(* implements non-volatile data using XML file and XML Server (max 4K) *)
FUNCTION_BLOCK FB_CX_NVData_XMLFile_4K
VAR_INPUT
	bEnable				: BOOL;		(* set TRUE to load and monitor XML data *)
	bReset				: BOOL;		(* set TRUE to reset error and re-start sequence *)
	bBackup				: BOOL;		(* set TRUE to write data to backup XML file *)
	bRestore			: BOOL;		(* set TRUE to restore data from backup XML file *)
	pSourceData			: POINTER TO BYTE;	(* pointer to source data structure *)
	nSourceBytes		: UDINT;		(* no of bytes in source data structure *)
	strXPath			: T_MaxString;	(* XPath for XML file *)
	strXMLPathFile		: T_MaxString;	(* XML file name, backup XML file will have '.bak' appended to the end *)
	tUpdateTime			: TIME;		(* update time to check for changes in memory *)
END_VAR
VAR_OUTPUT
	bNVDataInitOK		: BOOL;		(* TRUE = data loaded OK *)
	bFileWriteError		: BOOL;		(* TRUE = XML file write error *)
	bDataChanged		: BOOL;		(* TRUE = change of data detected *)
	nTotalChanges		: UDINT;	(* total number of data changes *)
END_VAR
VAR
	fbBackup			: R_TRIG;
	bBackupReq			: BOOL;
	fbRestore			: R_TRIG;
	bRestoreReq			: BOOL;

	eState				: E_CX_NVXMLState;
	fbDelayTimer		: TON;
	nRetries			: BYTE;
	fbReadXML			: FB_XmlSrvRead;
	fbMonitor			: FB_MemoryMonitor_4K;
	fbWriteXML			: FB_XmlSrvWrite;
	nOnlineChangeCount	: UDINT;
END_VAR
(*
-------------------------------------------------------------------------------------------------
Date		Version	Author	Comments
-------------------------------------------------------------------------------------------------
30/01/2015	3.00.00	PB		Initial release

-------------------------------------------------------------------------------------------------
*)

(* backup requested *)
fbBackup(CLK := bBackup);
IF fbBackup.Q = TRUE THEN

	bBackupReq := TRUE;
END_IF

(* restore requested *)
fbRestore(CLK := bRestore);
IF fbRestore.Q = TRUE THEN

	bRestoreReq := TRUE;
END_IF


CASE eState OF

	(* idle state *)
	E_CX_NVXML_IDLE:

		(* enabled*)
		IF bEnable = TRUE THEN

			(* update outputs *)
			bNVDataInitOK := FALSE;
			bFileWriteError := FALSE;

			eState := E_CX_NVXML_READXML;

		(* disabled *)
		ELSE

			(* reset outputs *)
			bNVDataInitOK := FALSE;
			bFileWriteError := FALSE;
			bDataChanged := FALSE;
			nTotalChanges := 0;

			(* reset event flags *)
			bBackupReq := FALSE;
			bRestoreReq := FALSE;
		END_IF


	(* read data *)
	E_CX_NVXML_READXML:

		(* read XML file *)
		fbReadXML(
			sNetId		:= '',
			ePath		:= PATH_GENERIC,
			nMode		:= XMLSRV_SKIPMISSING,
			pSymAddr	:= pSourceData,
			cbSymSize	:= nSourceBytes,
			sFilePath	:= strXMLPathFile,
			sXPath		:= strXPath,
			bExecute	:= TRUE,
			tTimeout	:= T#1s
		);

		(* XML read complete *)
		IF fbReadXML.bBusy = FALSE THEN

			(* XML read completed OK *)
			IF fbReadXML.bError = FALSE THEN

				(* XML file has been read at least once *)
				bNVDataInitOK := TRUE;

				eState := E_CX_NVXML_MONITOR;

			(* XML read error *)
			ELSE

				(* file access error *)
				IF fbReadXML.nErrId < 16#8000 THEN

					(* increment retry counter and wait for next read attempt *)
					nRetries := nRetries + 1;

					eState := E_CX_NVXML_RETRY;

				(* XML server error *)
				ELSE

					(* data has previously been read using XML Server *)
					IF bNVDataInitOK = TRUE THEN

						eState := E_CX_NVXML_MONITOR;

					(* data has not previously been read using XML Server *)
					ELSE

						eState := E_CX_NVXML_RESTORE;
					END_IF
				END_IF
			END_IF

			(* close off fbReadXML *)
			fbReadXML(bExecute := FALSE);
		END_IF


	(* restore backup data *)
	E_CX_NVXML_RESTORE:

		(* read XML backup file *)
		fbReadXML(
			sNetId		:= '',
			ePath		:= PATH_GENERIC,
			nMode		:= XMLSRV_SKIPMISSING,
			pSymAddr	:= pSourceData,
			cbSymSize	:= nSourceBytes,
			sFilePath	:= CONCAT(strXMLPathFile, '.bak'),
			sXPath		:= strXPath,
			bExecute	:= TRUE,
			tTimeout	:= T#1s
		);

		(* XML backup read complete *)
		IF fbReadXML.bBusy = FALSE THEN

			(* XML backup read completed OK *)
			IF fbReadXML.bError = FALSE THEN

				(* XML file has been read at least once *)
				bNVDataInitOK := TRUE;

				(* cancel restore request flag *)
				bRestoreReq := FALSE;

				eState := E_CX_NVXML_MONITOR;

			(* XML backup read error *)
			ELSE

				(* data has previously been read using XML Server *)
				IF bNVDataInitOK = TRUE THEN

					eState := E_CX_NVXML_MONITOR;

				(* data has not previously been read using XML Server *)
				ELSE

					eState := E_CX_NVXML_WRITEXML;
				END_IF
			END_IF

			(* close off fbReadXML *)
			fbReadXML(bExecute := FALSE);
		END_IF


	(* monitor state *)
	E_CX_NVXML_MONITOR:

		(* monitor specified data area for change of value *)
		fbMonitor(
			bEnable			:= TRUE,
			pSourceData		:= pSourceData,
			nSourceBytes	:= nSourceBytes,
			tUpdateTime		:= tUpdateTime,
			bDataChanged	=> bDataChanged,
			nTotalChanges	=> nTotalChanges
		);

		(* data monitoring disabled *)
		IF bEnable = FALSE THEN

			eState := E_CX_NVXML_IDLE;

		(* online program change, re-read data *)
		ELSIF  _AppInfo.OnlineChangeCnt <> nOnlineChangeCount THEN

			eState := E_CX_NVXML_READXML;

		(* restore from XML backup file requested *)
		ELSIF bRestoreReq = TRUE THEN

			eState := E_CX_NVXML_RESTORE;

		(* data has changed *)
		ELSIF bDataChanged = TRUE THEN

			eState := E_CX_NVXML_WRITEXML;

		(* write to XML backup file requested *)
		ELSIF bBackupReq = TRUE THEN

			eState := E_CX_NVXML_BACKUP;
		END_IF


	(* write data *)
	E_CX_NVXML_WRITEXML:

		(* write XML file *)
		fbWriteXML(
			sNetId		:= '',
			ePath		:= PATH_GENERIC,
			nMode		:= XMLSRV_ADDMISSING,
			pSymAddr	:= pSourceData,
			cbSymSize	:= nSourceBytes,
			sFilePath	:= strXMLPathFile,
			sXPath		:= strXPath,
			bExecute	:= TRUE,
			tTimeout	:= T#1s
		);

		(* XML file write complete *)
		IF fbWriteXML.bBusy = FALSE THEN

			(* XML file write completed OK *)
			IF fbWriteXML.bError = FALSE THEN

				(* cancel XML file write error *)
				bFileWriteError := FALSE;

				(* data has previously been read using XML Server *)
				IF bNVDataInitOK = TRUE THEN

					eState := E_CX_NVXML_MONITOR;

				(* data has not previously been read using XML Server *)
				ELSE

					eState := E_CX_NVXML_READXML;
				END_IF

			(* XML file write error *)
			ELSE

				(* unable to access file *)
				bFileWriteError := TRUE;

				(* return to monitor state *)
				eState := E_CX_NVXML_MONITOR;
			END_IF

			(* close off fbWriteXML *)
			fbWriteXML(bExecute := FALSE);
		END_IF


	(* write backup data *)
	E_CX_NVXML_BACKUP:

		(* write XML backup file *)
		fbWriteXML(
			sNetId		:= '',
			ePath		:= PATH_GENERIC,
			nMode		:= XMLSRV_ADDMISSING,
			pSymAddr	:= pSourceData,
			cbSymSize	:= nSourceBytes,
			sFilePath	:= CONCAT(strXMLPathFile, '.bak'),
			sXPath		:= strXPath,
			bExecute	:= TRUE,
			tTimeout	:= T#1s
		);

		(* XML backup file write complete *)
		IF fbWriteXML.bBusy = FALSE THEN

			(* XML backupfile write completed OK *)
			IF fbWriteXML.bError = FALSE THEN

				(* cancel save request flag *)
				bBackupReq := FALSE;

				(* return to monitor state *)
				eState := E_CX_NVXML_MONITOR;

			(* XML backupfile write error *)
			ELSE

				(* return to monitor state *)
				eState := E_CX_NVXML_MONITOR;
			END_IF

			(* close off fbWriteXML *)
			fbWriteXML(bExecute := FALSE);
		END_IF


	(* read failed *)
	E_CX_NVXML_RETRY:

		(* XML Server can take 3 seconds to start at boot-up, attempt to read XML file 5 times at startup with 1s between attempts before giving alarm *)

		(* data monitoring disabled *)
		IF bEnable = FALSE THEN

			eState := E_CX_NVXML_IDLE;

		(* 5 attempts to read file have failed *)
		ELSIF nRetries = 5 THEN

			eState := E_CX_NVXML_RESTORE;

		(* try to read XML file again *)
		ELSIF fbDelayTimer.Q = TRUE THEN

			eState := E_CX_NVXML_READXML;
		END_IF


(* unknown state *)
ELSE

	eState := E_CX_NVXML_IDLE;
END_CASE

(* re-read delay timer *)
fbDelayTimer(
	IN	:= eState = E_CX_NVXML_RETRY,
	PT	:= T#1s
);

(* log last value of online updates, allows online download to PLC program to be detected *)
nOnlineChangeCount :=  _AppInfo.OnlineChangeCnt;

END_FUNCTION_BLOCK

(* stored: Version 1.1.0.1
   POU FB_CX_NVData_XMLFile_4K: Id {ce23eed5-21f1-4654-b27c-0df6c7e41e45}, SpecialFunc None *)
